// TIA Portal V20 export
VAR_GLOBAL   // PLC tag table "Unit1Em7"
   "BA010AZCRPM04.14" AT %Q2013.4 : Bool;   // ELECTRODE NG BOX LOCK CYLINDER UP
   "BA010AZCRPM04.15" AT %Q2013.5 : Bool;   // ELECTRODE NG BOX LOCK CYLINDER DOWN
   "BA010AZCRBK05.06" AT %I1016.6 : Bool;   // ELECTRODE NG BOX LOCK CYLINDER DOWN
   "BA010AZCRBK05.16" AT %I1017.6 : Bool;   // ELECTRODE NG BOX LOCK CYLINDER UP
   "BA010AZCRBK07.04" AT %I1024.4 : Bool;   // ELECTRODE NG BOX FULL SENSOR
   "BA010AZCRSP506.03" AT %I3300.3 : Bool;   // ELECTRODE PASS KICKER DETECT SENSOR
   "BA010AZCRSP507.01" AT %I3350.1 : Bool;   // ELECTRODE DETECT COLOR SENSOR #1
   "BA010AZCRBK07.05" AT %I1024.5 : Bool;   // ELECTRODE NG BOX DETECT SENSOR
   "BA010AZCRSP507.02" AT %I3350.2 : Bool;   // ELECTRODE DETECT COLOR SENSOR #2
   "BA010AZCRSP507.00" AT %I3350.0 : Bool;   // ELECTRODE NG KICKER DETECT SENSOR
END_VAR
VAR_GLOBAL CONSTANT   // user constants
   U1EM7_NO_OF_AXES : USInt := 10;   // Starts with 1. E.g., the value 4 means that 4 axes exist.
   DR10_RatedTorque : LReal := 0.41;   // NgKickerAxisZ
   DR11_RatedTorque : LReal := 0.41;   // PassKickerAxisZ
   DR12_RatedTorque : LReal := 2.4;   // CutConveyorAxisB
   DR13_RatedTorque : LReal := 1.27;   // NgConveyorAxisB
   DR14_RatedTorque : LReal := 2.4;   // Stack1ConveyorAxisB
   DR15_RatedTorque : LReal := 3.2;   // Stack2ConveyorAxisB
   U1EM7_JOB01 : DInt := 1;
   U1EM7_JOB02 : DInt := 2;
   U1EM7_JOB03 : DInt := 3;
   U1EM7_JOB04 : DInt := 4;
   U1EM7_JOB05 : DInt := 5;
   U1EM7_JOB06 : DInt := 6;
   U1EM7_JOB07 : DInt := 7;
   U1EM7_JOB08 : DInt := 8;
   U1EM7_JOB09 : DInt := 9;
   U1EM7_JOB10 : DInt := 10;
   U1EM7_JOB11 : DInt := 11;
   U1EM7_JOB12 : DInt := 12;
   U1EM7_JOB13 : DInt := 13;
   U1EM7_JOB14 : DInt := 14;
   U1EM7_JOB15 : DInt := 15;
   U1EM7_JOB16 : DInt := 16;
   U1EM7_JOB17 : DInt := 17;
   U1EM7_JOB18 : DInt := 18;
   U1EM7_JOB19 : DInt := 19;
   U1EM7_JOB20 : DInt := 20;
   U1EM7_JOB21 : DInt := 21;
   U1EM7_JOB22 : DInt := 22;
   U1EM7_JOB23 : DInt := 23;
   U1EM7_JOB24 : DInt := 24;
   U1EM7_JOB25 : DInt := 25;
   U1EM7_JOB26 : DInt := 26;
   U1EM7_JOB27 : DInt := 27;
   U1EM7_JOB28 : DInt := 28;
   U1EM7_JOB29 : DInt := 29;
   U1EM7_JOB30 : DInt := 30;
   U1EM7_JOB31 : DInt := 31;
   U1EM7_JOB32 : DInt := 32;
   U1EM7_JOB33 : DInt := 33;
   U1EM7_JOB34 : DInt := 34;
   U1EM7_JOB35 : DInt := 35;
   U1EM7_JOB36 : DInt := 36;
   U1EM7_JOB37 : DInt := 37;
   U1EM7_JOB38 : DInt := 38;
   U1EM7_JOB39 : DInt := 39;
   U1EM7_JOB40 : DInt := 40;
   U1EM7_JOB41 : DInt := 41;
   U1EM7_JOB42 : DInt := 42;
   U1EM7_JOB43 : DInt := 43;
   U1EM7_JOB44 : DInt := 44;
   U1EM7_JOB45 : DInt := 45;
   U1EM7_JOB46 : DInt := 46;
   U1EM7_JOB47 : DInt := 47;
   U1EM7_JOB48 : DInt := 48;
   U1EM7_JOB49 : DInt := 49;
   U1EM7_JOB50 : DInt := 50;
END_VAR
